RoboDK station: PRACTICAL7.rdk

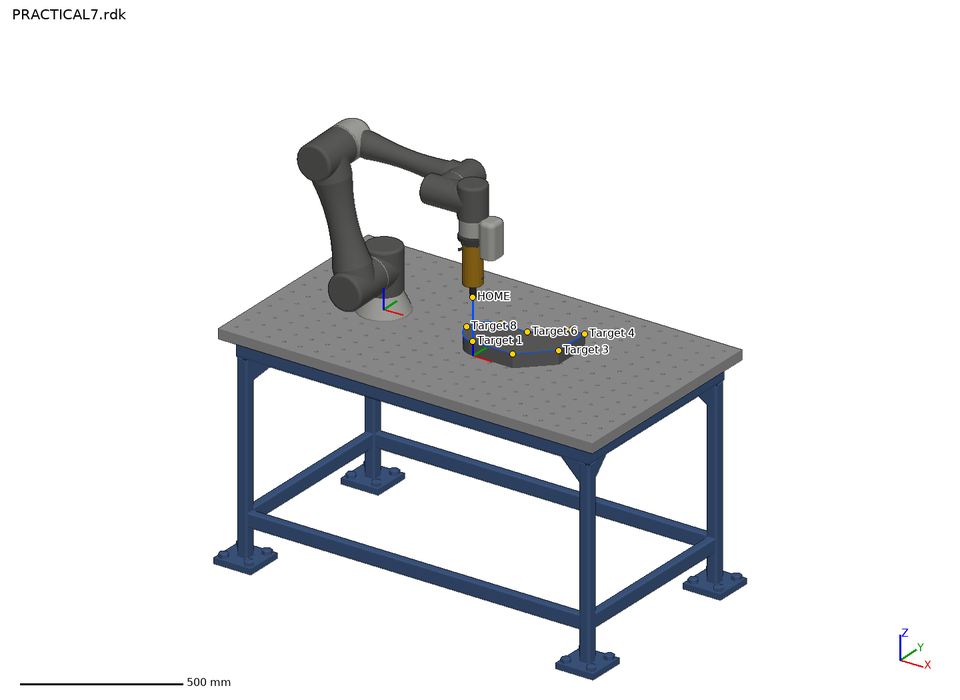
[picture v0: the station drawn from its stored meshes, robots at their saved joint values, targets as dots, program paths as lines]
Station PRACTICAL75 (saved by RoboDK 5.9.2). Poses are relative to the parent item; angles as X-Y-Z fixed-axis rotations.
  - frame TM5-900 Base at (0, 0, 0) mm
    - robot TM5-900: 6 axes, payload 4 kg, reach 900 mm, repeatability 0.1 mm, weight 30 kg
        modified DH rows (alpha deg, a mm, theta deg, d mm): 0, 0, 0, 145.2; 90, 0, 90, 0; 0, 429, 0, 0; 0, 411, -90, 122.3; -90, 0, 0, 106.5; 90, 0, 180, 114.15
        joint limits [-360, -180, -155, -180, -180, -270] to [360, 180, 155, 180, 180, 270]; home [0, 0, 90, -90, 90, 0]; saved at [1.726, -14.836, 109.127, -4.29, 90, 1.726]
      - tool ATI 9150-CDB-8-11-000 Deburring Tool (Spring), TCP at (0, 0, 215) mm, size 93.7 x 93.7 x 214.4 mm
  - object Table 1400x800x800mm at (0, 0, 0) mm, size 1420 x 820 x 800 mm, geometry from Table-1400x800x800mm.sld
  - frame Frame 2 at (410, -110, 0) mm
    - object random1 at (0, 0, 0) mm, size 325 x 240 x 50 mm, geometry from random1.step
    - target Target 1 (Cartesian target) at (0, 0, 49) mm, rotated rx 180 ry 0 rz 90 deg; joints [1.726, -8.549, 126.286, -27.737, 90, 1.726] of TM5-900
    - target Target 2 (Cartesian target) at (150, 0, 49) mm, rotated rx 180 ry 0 rz 90 deg; joints [1.261, 11.456, 105.687, -27.143, 90, 1.261] of TM5-900
    - target Target 3 (Cartesian target) at (250, 100, 49) mm, rotated rx 180 ry 0 rz 90 deg; joints [9.81, 22.604, 90.776, -23.38, 90, 9.81] of TM5-900
    - target Target 4 (Cartesian target) at (250, 239, 49) mm, rotated rx 180 ry 0 rz 90 deg; joints [21.538, 24.156, 88.525, -22.681, 90, 21.538] of TM5-900
    - target Target 5 (Cartesian target) at (200, 239, 49) mm, rotated rx 180 ry 0 rz 90 deg; joints [23.253, 18.055, 97.134, -25.189, 90, 23.253] of TM5-900
    - target Target 6 (Cartesian target) at (100, 149, 49) mm, rotated rx 180 ry 0 rz 90 deg; joints [18.207, 3.798, 114.543, -28.341, 90, 18.207] of TM5-900
    - target Target 7 (Cartesian target) at (0, 149, 49) mm, rotated rx 180 ry 0 rz 90 deg; joints [22.708, -10.512, 127.866, -27.354, 90, 22.708] of TM5-900
    - target Target 8 (Cartesian target) at (-75, 75, 49) mm, rotated rx 180 ry 0 rz 90 deg; joints [15.326, -23.496, 136.48, -22.983, 90, 15.326] of TM5-900
    - target HOME (Cartesian target) at (0, 0, 200) mm, rotated rx 180 ry 0 rz 90 deg; joints [1.726, -14.836, 109.127, -4.29, 90, 1.726] of TM5-900
  - program Prog1 (12 instructions, listed below)
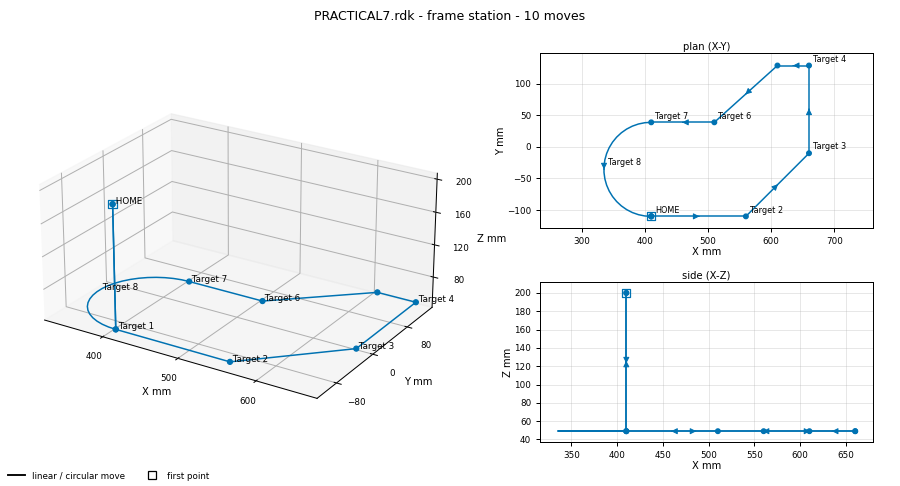
[picture p0: tool path of PRACTICAL7.rdk in frame station, 10 of 10 moves have a stored position in this frame; points joined in program order, loops and branches not executed]

--- program Prog1 (robot TM5-900) ---
  Set Ref.: Frame 2
  Set Tool: ATI 9150-CDB-8-11-000 Deburring Tool (Spring)
  MoveJ (HOME)
  MoveL (Target 1)
  MoveL (Target 2)
  MoveL (Target 3)
  MoveL (Target 4)
  MoveL (Target 5)
  MoveL (Target 6)
  MoveL (Target 7)
  MoveC (Target 8, Target 1)
  MoveL (HOME)
